(* PLC project Beremiz4Pico_BaseProject, Unknown NoName 1 *)
(* stored: creationDateTime 2020-08-28T21:59:35, modificationDateTime 2021-09-05T12:05:51 *)

CONFIGURATION config
  RESOURCE Resource1 ON PLC
    TASK PLCTask(INTERVAL := T#40ms, PRIORITY := 0);
  END_RESOURCE
END_CONFIGURATION
